// TIA Portal V20 export
FUNCTION_BLOCK "FB_IO_Device"   // FB4, LAD
{ S7_Optimized_Access := 'TRUE' }
// stored: MemoryReserve 100, SetENOAutomatically false
   VAR_INPUT
      Life_Trigger : Bool;
      Emergency_Stop_Release : Bool;
      Trigger_Read_Serial_Number_Entrace_Functional_Test : Bool;
      Trigger_Read_Serial_Number_Exit_Functional_Test : Bool;
      Selected_Voltage_220V : Bool;
      Selected_Voltage_127V : Bool;
      Carousel_Frequency_Inverter_Fail : Bool;
      Conveyor_Belt_Functional_Test_Inverter_Fail : Bool;
      In : "IO_Device_Inputs";
   END_VAR
   VAR_OUTPUT
      Start : Bool;
      Manual_Turn_On_Motor_Caroussel : Bool;
      Manual_Turn_On_Motor_Conveyor_Belt : Bool;
      Water_Foutain_Fail_Functional_Test : Bool;
      Select_Motor_Speed : SInt;
      Carousel_Voltage_Selection : SInt;
      Out : "IO_Device_Outputs";
   END_VAR
BEGIN

REGION Network 1
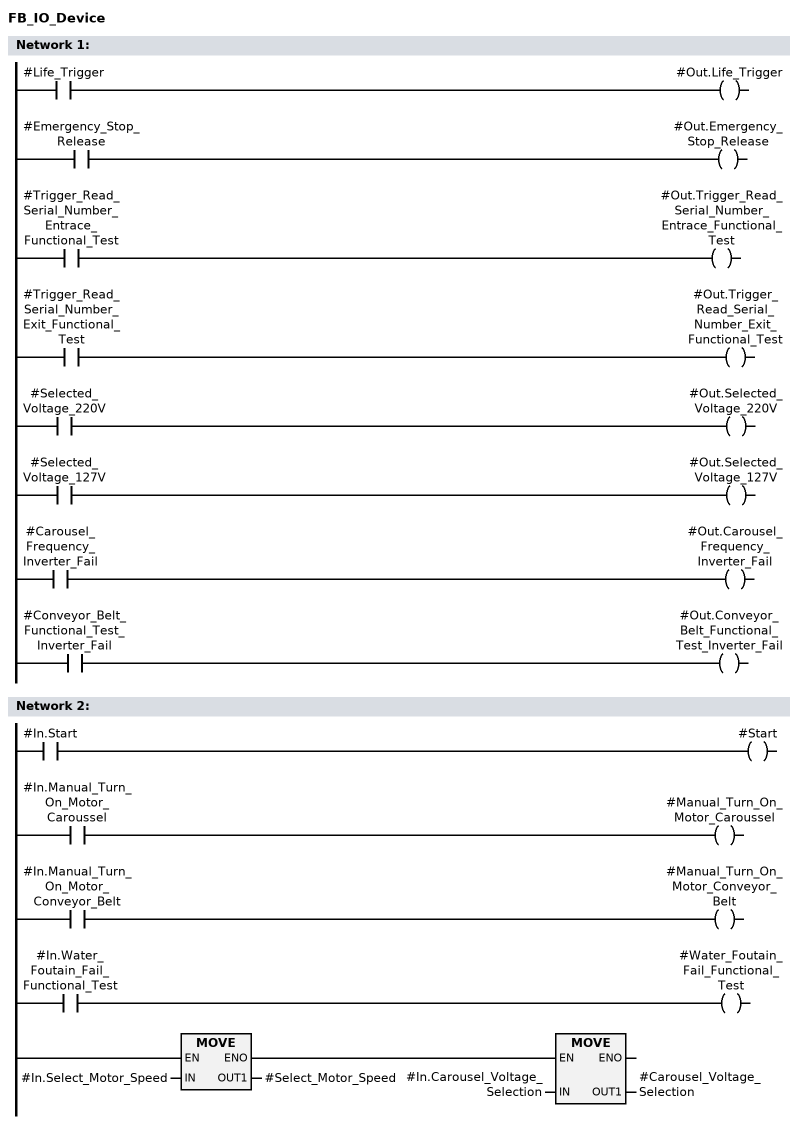
   RUNG wire#powerrail
      Contact( #Life_Trigger )
      Coil( #Out.Life_Trigger )
   END_RUNG
   RUNG wire#powerrail
      Contact( #Emergency_Stop_Release )
      Coil( #Out.Emergency_Stop_Release )
   END_RUNG
   RUNG wire#powerrail
      Contact( #Trigger_Read_Serial_Number_Entrace_Functional_Test )
      Coil( #Out.Trigger_Read_Serial_Number_Entrace_Functional_Test )
   END_RUNG
   RUNG wire#powerrail
      Contact( #Trigger_Read_Serial_Number_Exit_Functional_Test )
      Coil( #Out.Trigger_Read_Serial_Number_Exit_Functional_Test )
   END_RUNG
   RUNG wire#powerrail
      Contact( #Selected_Voltage_220V )
      Coil( #Out.Selected_Voltage_220V )
   END_RUNG
   RUNG wire#powerrail
      Contact( #Selected_Voltage_127V )
      Coil( #Out.Selected_Voltage_127V )
   END_RUNG
   RUNG wire#powerrail
      Contact( #Carousel_Frequency_Inverter_Fail )
      Coil( #Out.Carousel_Frequency_Inverter_Fail )
   END_RUNG
   RUNG wire#powerrail
      Contact( #Conveyor_Belt_Functional_Test_Inverter_Fail )
      Coil( #Out.Conveyor_Belt_Functional_Test_Inverter_Fail )
   END_RUNG
   // the same network as SCL:
   #Out.Life_Trigger := #Life_Trigger;
   #Out.Emergency_Stop_Release := #Emergency_Stop_Release;
   #Out.Trigger_Read_Serial_Number_Entrace_Functional_Test := #Trigger_Read_Serial_Number_Entrace_Functional_Test;
   #Out.Trigger_Read_Serial_Number_Exit_Functional_Test := #Trigger_Read_Serial_Number_Exit_Functional_Test;
   #Out.Selected_Voltage_220V := #Selected_Voltage_220V;
   #Out.Selected_Voltage_127V := #Selected_Voltage_127V;
   #Out.Carousel_Frequency_Inverter_Fail := #Carousel_Frequency_Inverter_Fail;
   #Out.Conveyor_Belt_Functional_Test_Inverter_Fail := #Conveyor_Belt_Functional_Test_Inverter_Fail;
END_REGION

REGION Network 2
   RUNG wire#powerrail
      Contact( #In.Start )
      Coil( #Start )
   END_RUNG
   RUNG wire#powerrail
      Contact( #In.Manual_Turn_On_Motor_Caroussel )
      Coil( #Manual_Turn_On_Motor_Caroussel )
   END_RUNG
   RUNG wire#powerrail
      Contact( #In.Manual_Turn_On_Motor_Conveyor_Belt )
      Coil( #Manual_Turn_On_Motor_Conveyor_Belt )
   END_RUNG
   RUNG wire#powerrail
      Contact( #In.Water_Foutain_Fail_Functional_Test )
      Coil( #Water_Foutain_Fail_Functional_Test )
   END_RUNG
   RUNG wire#powerrail
      Move(in := #In.Select_Motor_Speed, out1 => #Select_Motor_Speed)
      Move(in := #In.Carousel_Voltage_Selection, out1 => #Carousel_Voltage_Selection)
   END_RUNG
   // the same network as SCL:
   #Start := #In.Start;
   #Manual_Turn_On_Motor_Caroussel := #In.Manual_Turn_On_Motor_Caroussel;
   #Manual_Turn_On_Motor_Conveyor_Belt := #In.Manual_Turn_On_Motor_Conveyor_Belt;
   #Water_Foutain_Fail_Functional_Test := #In.Water_Foutain_Fail_Functional_Test;
   #Select_Motor_Speed := #In.Select_Motor_Speed;
   #Carousel_Voltage_Selection := #In.Carousel_Voltage_Selection;
END_REGION
END_FUNCTION_BLOCK
